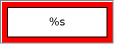
VISUALIZATION Visu_StanMaszyny_AktualyStan  // 114x44
VAR_IN_OUT
	bNacisniety								: BOOL;
END_VAR
VAR_INPUT
	stVisuStan								: DUT_StanMaszyny_VISU_Stan;
END_VAR
    RoundedRectangle (2,2 110x40), invisible if: not stVisuStan.bAktywny
    RoundedRectangle (7,7 100x30), "%s", text variable: stVisuStan.sNazwa, colour variable: 16#FF000000 OR (16#FF000000 OR (stVisuStan.dwKolorTla))
        OnMouseDown: execute {
            //IF (stVisuStan.bAktywny) THEN
            	bNacisniety := stVisuStan.bAktywny AND TRUE;
            //END_IF
        }
END_VISUALIZATION

(* stored: Version 1.1.0.1, ProductVersion 3.1.4024.11
   Visu Visu_StanMaszyny_AktualyStan: Id {320aad0e-094f-4109-98e0-1c01f37d6189} *)
